_CFC_ (* Continuous Function Chart, elements in execution order *)
#0 OR(changeValueWithoutPower, ctrlVoltage)
#1 AND(#0, enable)
#2 OR(byError.3, byError.4)
#3 AND(#2, TON_DOST.Q)
#4 OR(reset, #3)
#5 fb_HVACAI:FB_HVACAnalogInput(EN: #1, eHVACDataSecurityType_Idle, FALSE, rawValue, tTaskCycleTime, tTaskCycleTime, enableLimitCtrl, ctrlVoltage, #4, iHighRange, iLowRange, highRange, lowRange, highLimit, lowLimit, filterTime, offset)
#6 presentValue <= #5.out 1
#7 byState <= #5.out 2
#8 byError <= #5.out 8
#9 I_GT:ISTOK_GT(dost: TRUE, x: #5.out 1, ust: highLimit, shkal: -, gist: 1)
#10 I_LT:ISTOK_LT(dost: TRUE, x: #5.out 1, ust: lowLimit, shkal: -, gist: 1)
#11 OR(#9.Xb, #10.Xm)
#12 TON_DOST:TON(IN: NOT #11, PT: T#10s)
#13 delay:TON(IN: ctrlVoltage, PT: delayEnable)
#14 AND(TON_DOST.Q, #13.Q)
#15 RS_AI:RS(SET: #14, RESET1: error)
#16 reliability <= #15.Q1
#17 >(byError, 0)
#18 OR(#17, NOT ctrlVoltage)
#19 error <= #18
_END_CFC_
END_FUNCTION_BLOCK

(* POU Lib/ISTOK_GT, CFC *)
FUNCTION_BLOCK ISTOK_GT
VAR_INPUT
	dost: BOOL;
	x: REAL;
	ust: REAL;
	shkal: REAL;
	gist: REAL;
END_VAR
VAR_OUTPUT
	Xb: BOOL;
	XbN: BOOL;
END_VAR
VAR
	rs_gt: RS;
END_VAR
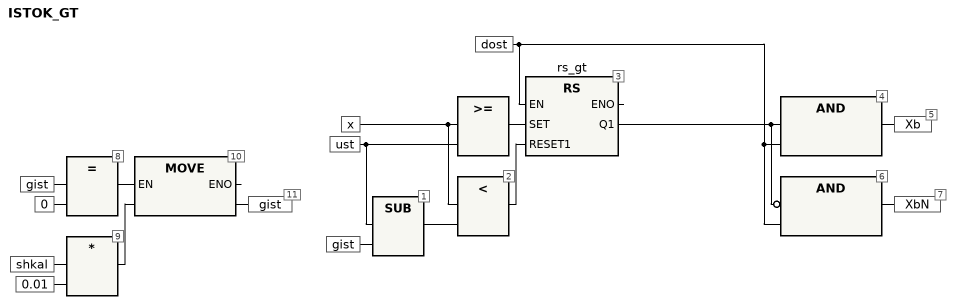
_CFC_ (* Continuous Function Chart, elements in execution order *)
#0 >=(x, ust)
#1 SUB(ust, gist)
#2 <(x, #1)
#3 rs_gt:RS(EN: dost, SET: #0, RESET1: #2)
#4 AND(#3.Q1, dost)
#5 Xb <= #4
#6 AND(NOT #3.Q1, dost)
#7 XbN <= #6
#8 =(gist, 0)
#9 *(shkal, 0.01)
#10 MOVE(EN: #8, #9)
#11 gist <= #10
_END_CFC_
END_FUNCTION_BLOCK

(* POU Lib/ISTOK_LT, CFC *)
FUNCTION_BLOCK ISTOK_LT
VAR_INPUT
	dost: BOOL;
	x: REAL;
	ust: REAL;
	shkal: REAL;
	gist: REAL;
END_VAR
VAR_OUTPUT
	Xm: BOOL;
	XmN: BOOL;
END_VAR
VAR
	rs_lt: RS;
END_VAR
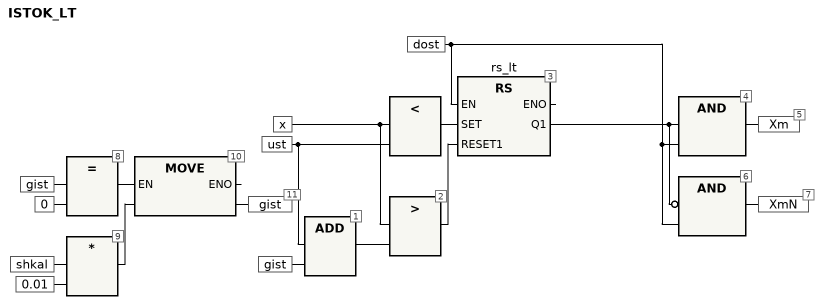
_CFC_ (* Continuous Function Chart, elements in execution order *)
#0 <(x, ust)
#1 ADD(ust, gist)
#2 >(x, #1)
#3 rs_lt:RS(EN: dost, SET: #0, RESET1: #2)
#4 AND(#3.Q1, dost)
#5 Xm <= #4
#6 AND(NOT #3.Q1, dost)
#7 XmN <= #6
#8 =(gist, 0)
#9 *(shkal, 0.01)
#10 MOVE(EN: #8, #9)
#11 gist <= #10
_END_CFC_
END_FUNCTION_BLOCK

(* POU Input/AI/TE1, CFC *)
PROGRAM TE1
VAR
	fb_TE1: ISTOK_ANALOGVH;
	ofset: REAL;
	fb_SCHU_P2_4_TE1_B_UST_MYAG_REG: ISTOK_GT;
	fb_SCHU_P2_4_TE1_B_UST_SEZ_LETO: ISTOK_GT;
	I_GT_TE: ISTOK_GT;
	I_LT_TE: ISTOK_LT;
	TON_DOST: TON;
END_VAR
VAR (* helpers for the ST form of the networks *)
	_t75 : REAL;
END_VAR
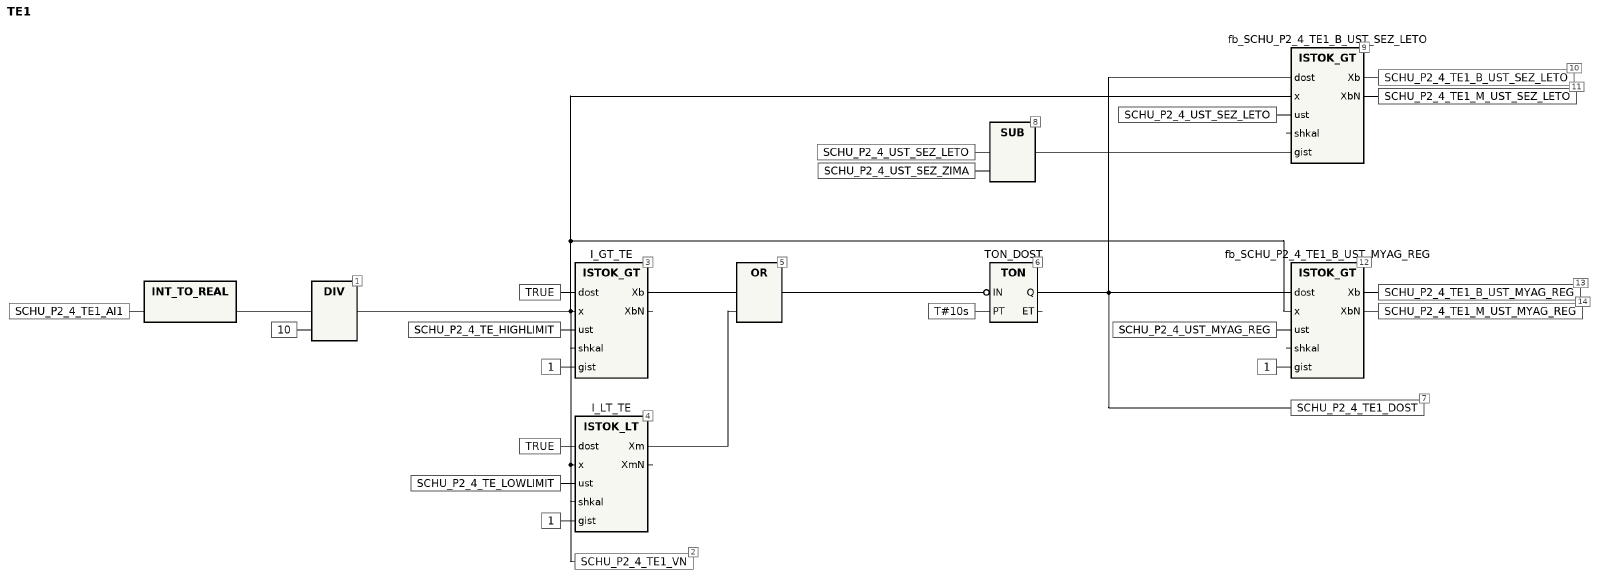
_CFC_ (* Continuous Function Chart, elements in execution order *)
#0 INT_TO_REAL(SCHU_P2_4_TE1_AI1)
#1 DIV(#0, 10)
#2 SCHU_P2_4_TE1_VN <= #1
#3 I_GT_TE:ISTOK_GT(dost: TRUE, x: #1, ust: SCHU_P2_4_TE_HIGHLIMIT, shkal: -, gist: 1)
#4 I_LT_TE:ISTOK_LT(dost: TRUE, x: #1, ust: SCHU_P2_4_TE_LOWLIMIT, shkal: -, gist: 1)
#5 OR(#3.Xb, #4.Xm)
#6 TON_DOST:TON(IN: NOT #5, PT: T#10s)
#7 SCHU_P2_4_TE1_DOST <= #6.Q
#8 SUB(SCHU_P2_4_UST_SEZ_LETO, SCHU_P2_4_UST_SEZ_ZIMA)
#9 fb_SCHU_P2_4_TE1_B_UST_SEZ_LETO:ISTOK_GT(dost: #6.Q, x: #1, ust: SCHU_P2_4_UST_SEZ_LETO, shkal: -, gist: #8)
#10 SCHU_P2_4_TE1_B_UST_SEZ_LETO <= #9.Xb
#11 SCHU_P2_4_TE1_M_UST_SEZ_LETO <= #9.XbN
#12 fb_SCHU_P2_4_TE1_B_UST_MYAG_REG:ISTOK_GT(dost: #6.Q, x: #1, ust: SCHU_P2_4_UST_MYAG_REG, shkal: -, gist: 1)
#13 SCHU_P2_4_TE1_B_UST_MYAG_REG <= #12.Xb
#14 SCHU_P2_4_TE1_M_UST_MYAG_REG <= #12.XbN
_END_CFC_
(* the same logic as Structured Text *)
_t75 := INT_TO_REAL(SCHU_P2_4_TE1_AI1) / 10;
SCHU_P2_4_TE1_VN := _t75;
I_GT_TE(dost := TRUE, x := _t75, ust := SCHU_P2_4_TE_HIGHLIMIT, gist := 1);
I_LT_TE(dost := TRUE, x := _t75, ust := SCHU_P2_4_TE_LOWLIMIT, gist := 1);
TON_DOST(IN := NOT (I_GT_TE.Xb OR I_LT_TE.Xm), PT := T#10s);
SCHU_P2_4_TE1_DOST := TON_DOST.Q;
fb_SCHU_P2_4_TE1_B_UST_SEZ_LETO(dost := TON_DOST.Q, x := _t75, ust := SCHU_P2_4_UST_SEZ_LETO, gist := SCHU_P2_4_UST_SEZ_LETO - SCHU_P2_4_UST_SEZ_ZIMA);
SCHU_P2_4_TE1_B_UST_SEZ_LETO := fb_SCHU_P2_4_TE1_B_UST_SEZ_LETO.Xb;
SCHU_P2_4_TE1_M_UST_SEZ_LETO := fb_SCHU_P2_4_TE1_B_UST_SEZ_LETO.XbN;
fb_SCHU_P2_4_TE1_B_UST_MYAG_REG(dost := TON_DOST.Q, x := _t75, ust := SCHU_P2_4_UST_MYAG_REG, gist := 1);
SCHU_P2_4_TE1_B_UST_MYAG_REG := fb_SCHU_P2_4_TE1_B_UST_MYAG_REG.Xb;
SCHU_P2_4_TE1_M_UST_MYAG_REG := fb_SCHU_P2_4_TE1_B_UST_MYAG_REG.XbN;
END_PROGRAM

(* POU Input/AI/TE2, CFC *)
PROGRAM TE2
VAR
	TE2_YST: REAL;
	fb_TE2: ISTOK_ANALOGVH;
	ofset: REAL;
	fb_SCHU_P2_4_TE2_M_ZASCH: ISTOK_LT;
	fb_SCHU_P2_4_TE2_M_UST: ISTOK_LT;
	I_GT_TE: ISTOK_GT;
	I_LT_TE: ISTOK_LT;
	TON_DOST: TON;
END_VAR
VAR (* helpers for the ST form of the networks *)
	_t112 : REAL;
END_VAR
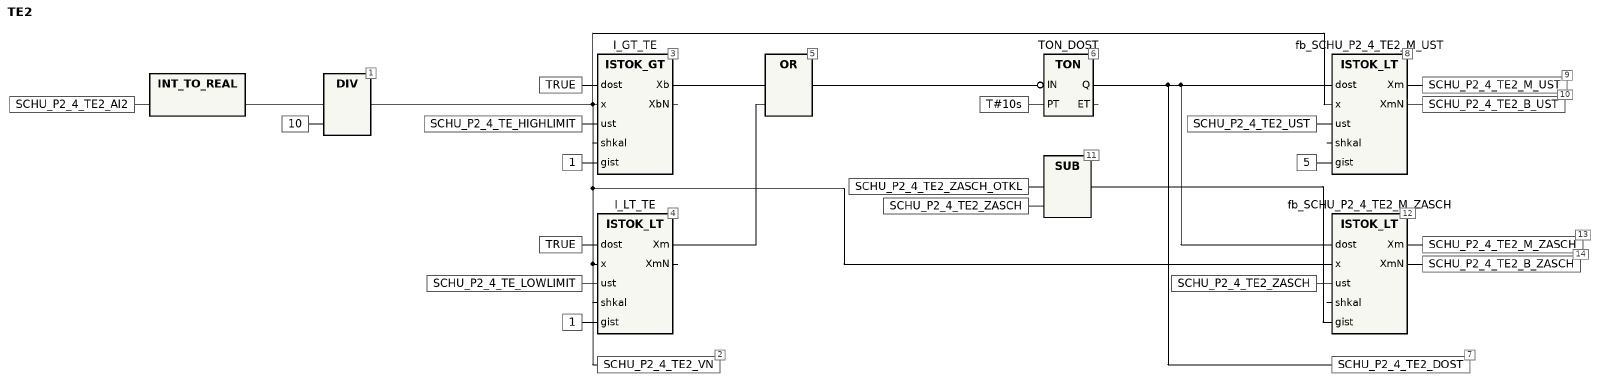
